SYSTEM temexdmodluyben
  (* Version 1.0, Author, 4DIAC-Consortium *)
  APPLICATION App1_ProdRateandPressure
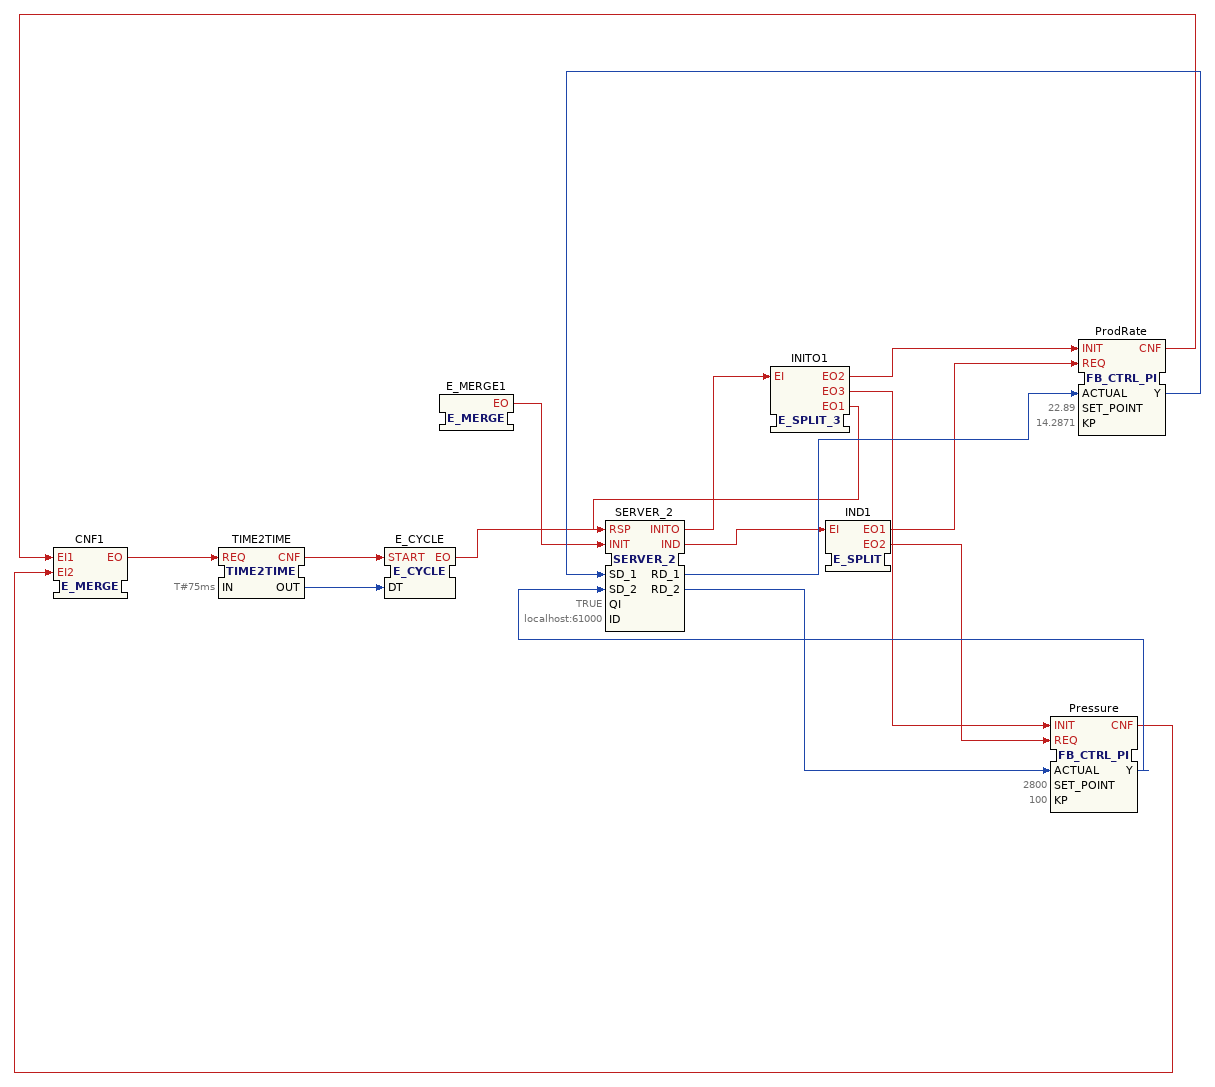
    FBS
      ProdRate : FB_CTRL_PI(SET_POINT := 22.89, KP := 14.2871);
      E_CYCLE : E_CYCLE;
      TIME2TIME : TIME2TIME(IN := T#75ms);
      SERVER_2 : SERVER_2(QI := TRUE, ID := localhost:61000);
      Pressure : FB_CTRL_PI(SET_POINT := 2800, KP := 100);
      INITO1 : E_SPLIT_3;
      IND1 : E_SPLIT;
      CNF1 : E_MERGE;
      E_MERGE1 : E_MERGE;
    END_FBS
    EVENT_CONNECTIONS
      TIME2TIME.CNF TO E_CYCLE.START;
      E_CYCLE.EO TO SERVER_2.RSP;
      SERVER_2.INITO TO INITO1.EI;
      INITO1.EO2 TO ProdRate.INIT;
      INITO1.EO3 TO Pressure.INIT;
      INITO1.EO1 TO SERVER_2.RSP;
      SERVER_2.IND TO IND1.EI;
      IND1.EO1 TO ProdRate.REQ;
      IND1.EO2 TO Pressure.REQ;
      ProdRate.CNF TO CNF1.EI1;
      Pressure.CNF TO CNF1.EI2;
      CNF1.EO TO TIME2TIME.REQ;
      E_MERGE1.EO TO SERVER_2.INIT;
    END_CONNECTIONS
    DATA_CONNECTIONS
      TIME2TIME.OUT TO E_CYCLE.DT;
      SERVER_2.RD_1 TO ProdRate.ACTUAL;
      SERVER_2.RD_2 TO Pressure.ACTUAL;
      ProdRate.Y TO SERVER_2.SD_1;
      Pressure.Y TO SERVER_2.SD_2;
    END_CONNECTIONS
  END_APPLICATION
  APPLICATION App2_StripperTemperatureandReactorTemperature
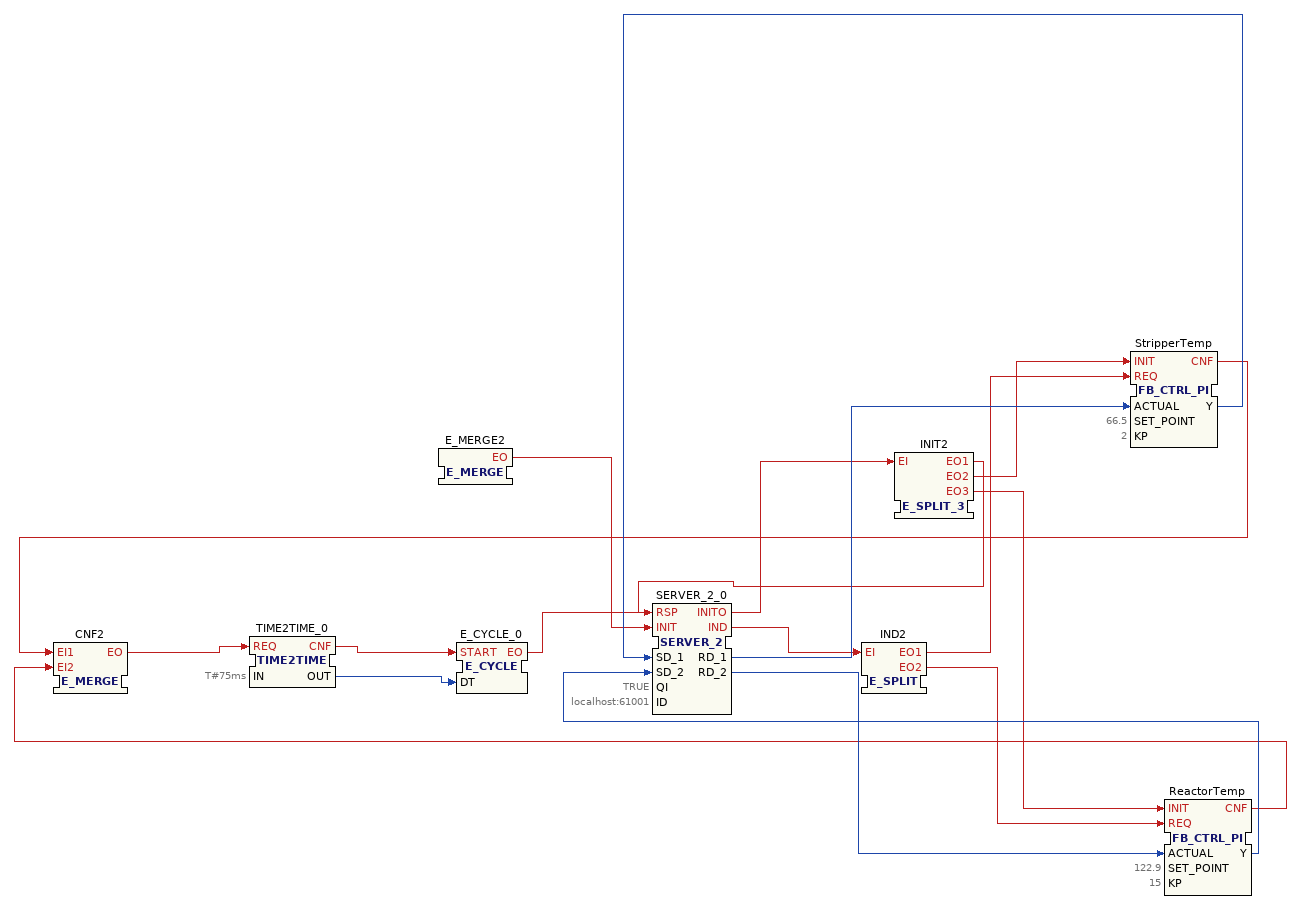
    FBS
      StripperTemp : FB_CTRL_PI(SET_POINT := 66.5, KP := 2);
      E_CYCLE_0 : E_CYCLE;
      TIME2TIME_0 : TIME2TIME(IN := T#75ms);
      SERVER_2_0 : SERVER_2(QI := TRUE, ID := localhost:61001);
      ReactorTemp : FB_CTRL_PI(SET_POINT := 122.9, KP := 15);
      CNF2 : E_MERGE;
      IND2 : E_SPLIT;
      INIT2 : E_SPLIT_3;
      E_MERGE2 : E_MERGE;
    END_FBS
    EVENT_CONNECTIONS
      E_CYCLE_0.EO TO SERVER_2_0.RSP;
      TIME2TIME_0.CNF TO E_CYCLE_0.START;
      SERVER_2_0.INITO TO INIT2.EI;
      INIT2.EO1 TO SERVER_2_0.RSP;
      INIT2.EO2 TO StripperTemp.INIT;
      INIT2.EO3 TO ReactorTemp.INIT;
      SERVER_2_0.IND TO IND2.EI;
      IND2.EO1 TO StripperTemp.REQ;
      IND2.EO2 TO ReactorTemp.REQ;
      StripperTemp.CNF TO CNF2.EI1;
      ReactorTemp.CNF TO CNF2.EI2;
      CNF2.EO TO TIME2TIME_0.REQ;
      E_MERGE2.EO TO SERVER_2_0.INIT;
    END_CONNECTIONS
    DATA_CONNECTIONS
      TIME2TIME_0.OUT TO E_CYCLE_0.DT;
      StripperTemp.Y TO SERVER_2_0.SD_1;
      SERVER_2_0.RD_1 TO StripperTemp.ACTUAL;
      SERVER_2_0.RD_2 TO ReactorTemp.ACTUAL;
      ReactorTemp.Y TO SERVER_2_0.SD_2;
    END_CONNECTIONS
  END_APPLICATION
  APPLICATION App3_StripperLevelandSeparatorLevel
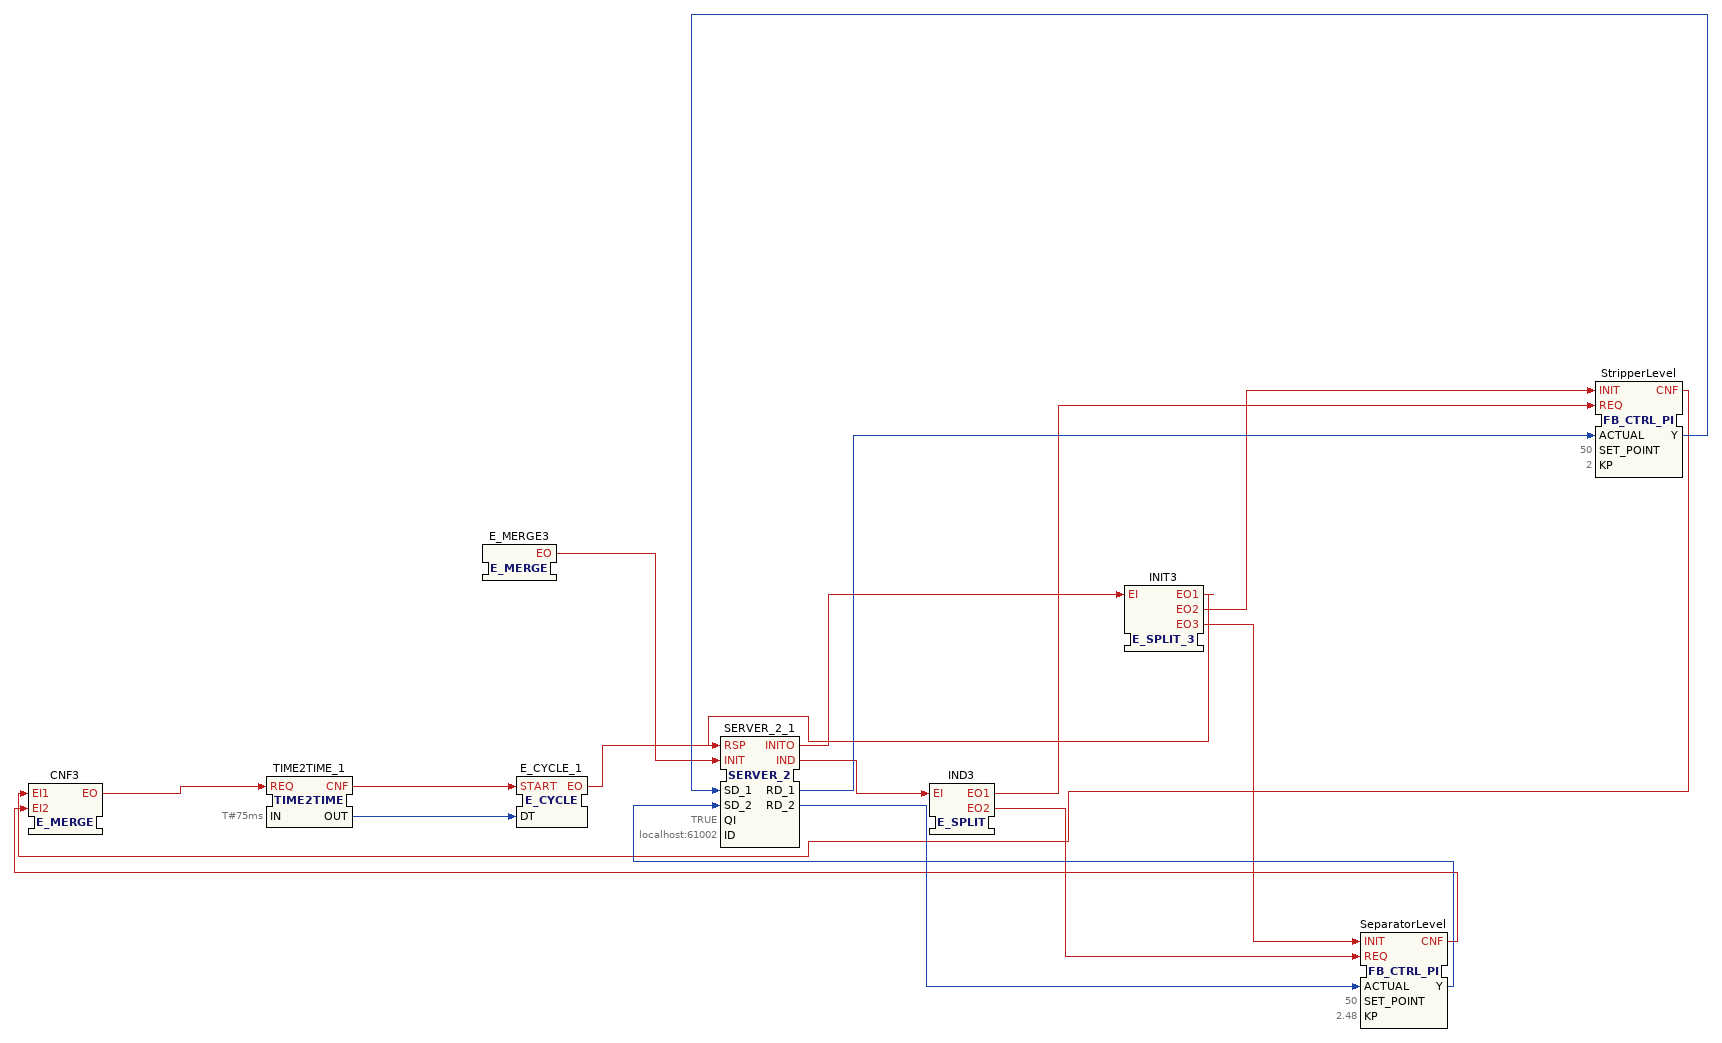
    FBS
      StripperLevel : FB_CTRL_PI(SET_POINT := 50, KP := 2);
      E_CYCLE_1 : E_CYCLE;
      TIME2TIME_1 : TIME2TIME(IN := T#75ms);
      SERVER_2_1 : SERVER_2(QI := TRUE, ID := localhost:61002);
      SeparatorLevel : FB_CTRL_PI(SET_POINT := 50, KP := 2.48);
      INIT3 : E_SPLIT_3;
      IND3 : E_SPLIT;
      CNF3 : E_MERGE;
      E_MERGE3 : E_MERGE;
    END_FBS
    EVENT_CONNECTIONS
      E_CYCLE_1.EO TO SERVER_2_1.RSP;
      TIME2TIME_1.CNF TO E_CYCLE_1.START;
      SERVER_2_1.INITO TO INIT3.EI;
      INIT3.EO1 TO SERVER_2_1.RSP;
      INIT3.EO2 TO StripperLevel.INIT;
      INIT3.EO3 TO SeparatorLevel.INIT;
      SERVER_2_1.IND TO IND3.EI;
      IND3.EO1 TO StripperLevel.REQ;
      IND3.EO2 TO SeparatorLevel.REQ;
      CNF3.EO TO TIME2TIME_1.REQ;
      StripperLevel.CNF TO CNF3.EI1;
      SeparatorLevel.CNF TO CNF3.EI2;
      E_MERGE3.EO TO SERVER_2_1.INIT;
    END_CONNECTIONS
    DATA_CONNECTIONS
      TIME2TIME_1.OUT TO E_CYCLE_1.DT;
      StripperLevel.Y TO SERVER_2_1.SD_1;
      SERVER_2_1.RD_1 TO StripperLevel.ACTUAL;
      SERVER_2_1.RD_2 TO SeparatorLevel.ACTUAL;
      SeparatorLevel.Y TO SERVER_2_1.SD_2;
    END_CONNECTIONS
  END_APPLICATION
  APPLICATION App4_ReactorLevel
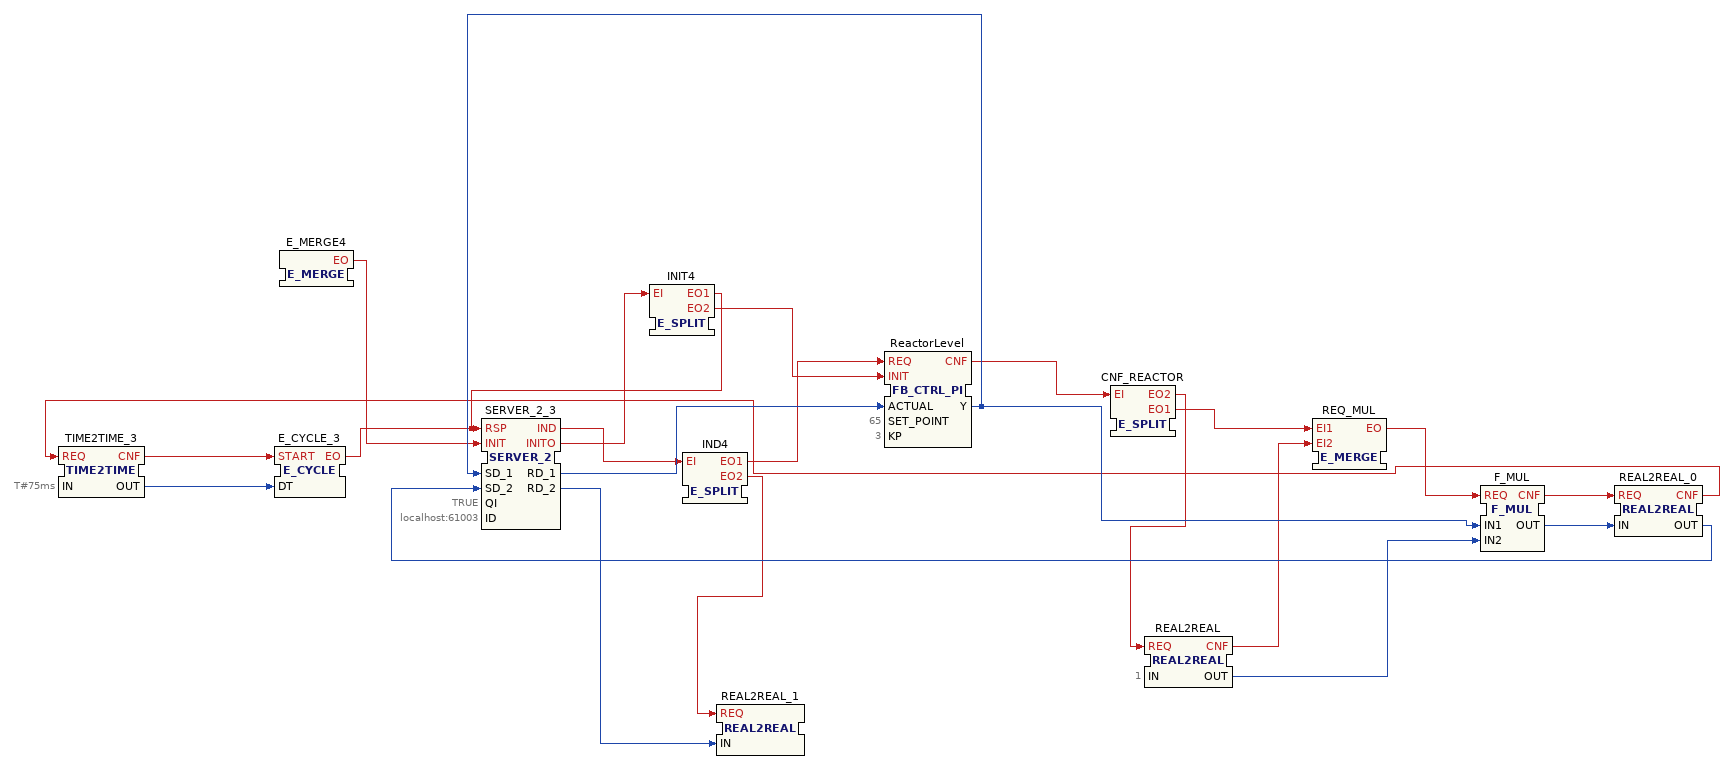
    FBS
      ReactorLevel : FB_CTRL_PI(SET_POINT := 65, KP := 3);
      E_CYCLE_3 : E_CYCLE;
      TIME2TIME_3 : TIME2TIME(IN := T#75ms);
      SERVER_2_3 : SERVER_2(QI := TRUE, ID := localhost:61003);
      F_MUL : F_MUL;
      REAL2REAL : REAL2REAL(IN := 1);
      REAL2REAL_0 : REAL2REAL;
      REAL2REAL_1 : REAL2REAL;
      IND4 : E_SPLIT;
      INIT4 : E_SPLIT;
      REQ_MUL : E_MERGE;
      CNF_REACTOR : E_SPLIT;
      E_MERGE4 : E_MERGE;
    END_FBS
    EVENT_CONNECTIONS
      E_CYCLE_3.EO TO SERVER_2_3.RSP;
      TIME2TIME_3.CNF TO E_CYCLE_3.START;
      F_MUL.CNF TO REAL2REAL_0.REQ;
      REAL2REAL_0.CNF TO TIME2TIME_3.REQ;
      SERVER_2_3.IND TO IND4.EI;
      IND4.EO1 TO ReactorLevel.REQ;
      IND4.EO2 TO REAL2REAL_1.REQ;
      SERVER_2_3.INITO TO INIT4.EI;
      INIT4.EO1 TO SERVER_2_3.RSP;
      INIT4.EO2 TO ReactorLevel.INIT;
      ReactorLevel.CNF TO CNF_REACTOR.EI;
      CNF_REACTOR.EO2 TO REAL2REAL.REQ;
      CNF_REACTOR.EO1 TO REQ_MUL.EI1;
      REAL2REAL.CNF TO REQ_MUL.EI2;
      REQ_MUL.EO TO F_MUL.REQ;
      E_MERGE4.EO TO SERVER_2_3.INIT;
    END_CONNECTIONS
    DATA_CONNECTIONS
      TIME2TIME_3.OUT TO E_CYCLE_3.DT;
      ReactorLevel.Y TO SERVER_2_3.SD_1;
      SERVER_2_3.RD_1 TO ReactorLevel.ACTUAL;
      ReactorLevel.Y TO F_MUL.IN1;
      REAL2REAL.OUT TO F_MUL.IN2;
      F_MUL.OUT TO REAL2REAL_0.IN;
      REAL2REAL_0.OUT TO SERVER_2_3.SD_2;
      SERVER_2_3.RD_2 TO REAL2REAL_1.IN;
    END_CONNECTIONS
  END_APPLICATION
  APPLICATION App5_yAandyB
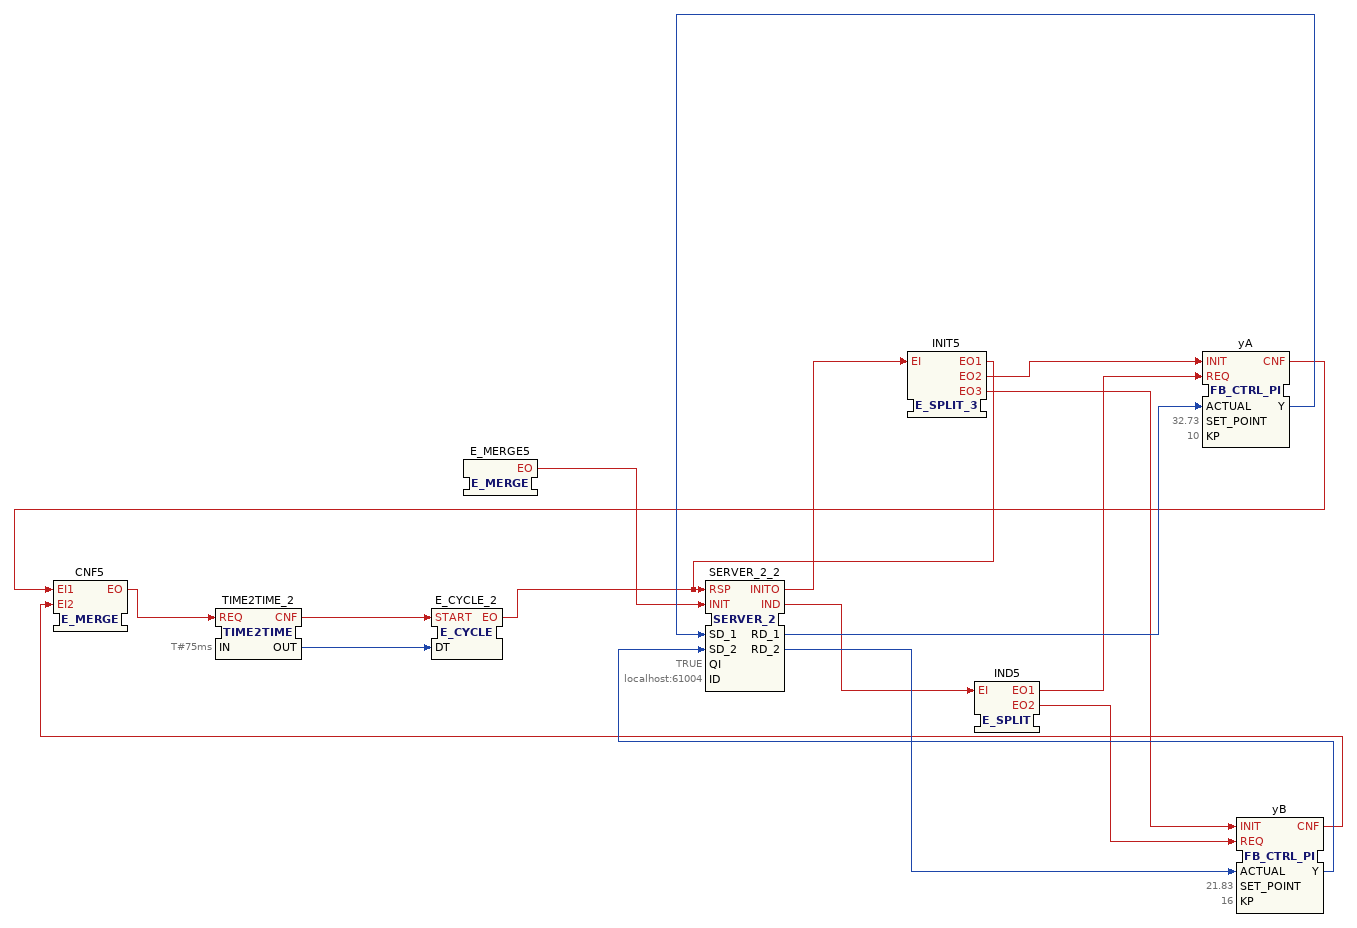
    FBS
      yA : FB_CTRL_PI(SET_POINT := 32.73, KP := 10);
      E_CYCLE_2 : E_CYCLE;
      TIME2TIME_2 : TIME2TIME(IN := T#75ms);
      SERVER_2_2 : SERVER_2(QI := TRUE, ID := localhost:61004);
      yB : FB_CTRL_PI(SET_POINT := 21.83, KP := 16);
      INIT5 : E_SPLIT_3;
      IND5 : E_SPLIT;
      CNF5 : E_MERGE;
      E_MERGE5 : E_MERGE;
    END_FBS
    EVENT_CONNECTIONS
      E_CYCLE_2.EO TO SERVER_2_2.RSP;
      TIME2TIME_2.CNF TO E_CYCLE_2.START;
      SERVER_2_2.INITO TO INIT5.EI;
      INIT5.EO1 TO SERVER_2_2.RSP;
      INIT5.EO2 TO yA.INIT;
      INIT5.EO3 TO yB.INIT;
      SERVER_2_2.IND TO IND5.EI;
      IND5.EO1 TO yA.REQ;
      IND5.EO2 TO yB.REQ;
      CNF5.EO TO TIME2TIME_2.REQ;
      yA.CNF TO CNF5.EI1;
      yB.CNF TO CNF5.EI2;
      E_MERGE5.EO TO SERVER_2_2.INIT;
    END_CONNECTIONS
    DATA_CONNECTIONS
      TIME2TIME_2.OUT TO E_CYCLE_2.DT;
      yA.Y TO SERVER_2_2.SD_1;
      SERVER_2_2.RD_1 TO yA.ACTUAL;
      SERVER_2_2.RD_2 TO yB.ACTUAL;
      yB.Y TO SERVER_2_2.SD_2;
    END_CONNECTIONS
  END_APPLICATION
  DEVICE FORTE_PC : FORTE_PC(MGR_ID := "localhost:61499")
    {SET_ATTRIBUTE(Profile, HOLOBLOC)}
    RESOURCE EMB_RES : EMB_RES
      FBS
        ProdRate : FB_CTRL_PI(SET_POINT := 22.89, KP := 14.2871);
        E_CYCLE : E_CYCLE;
        TIME2TIME : TIME2TIME(IN := T#75ms);
        SERVER_2 : SERVER_2(QI := TRUE, ID := localhost:61000);
        Pressure : FB_CTRL_PI(SET_POINT := 2800, KP := 100);
        StripperTemp : FB_CTRL_PI(SET_POINT := 66.5, KP := 2);
        E_CYCLE_0 : E_CYCLE;
        TIME2TIME_0 : TIME2TIME(IN := T#75ms);
        SERVER_2_0 : SERVER_2(QI := TRUE, ID := localhost:61001);
        ReactorTemp : FB_CTRL_PI(SET_POINT := 122.9, KP := 15);
        ReactorLevel : FB_CTRL_PI(SET_POINT := 65, KP := 3);
        E_CYCLE_3 : E_CYCLE;
        TIME2TIME_3 : TIME2TIME(IN := T#75ms);
        SERVER_2_3 : SERVER_2(QI := TRUE, ID := localhost:61003);
        F_MUL : F_MUL;
        REAL2REAL : REAL2REAL(IN := 1);
        REAL2REAL_0 : REAL2REAL;
        REAL2REAL_1 : REAL2REAL;
        yA : FB_CTRL_PI(SET_POINT := 32.73, KP := 10);
        E_CYCLE_2 : E_CYCLE;
        TIME2TIME_2 : TIME2TIME(IN := T#75ms);
        SERVER_2_2 : SERVER_2(QI := TRUE, ID := localhost:61004);
        yB : FB_CTRL_PI(SET_POINT := 21.83, KP := 16);
        StripperLevel : FB_CTRL_PI(SET_POINT := 50, KP := 2);
        E_CYCLE_1 : E_CYCLE;
        TIME2TIME_1 : TIME2TIME(IN := T#75ms);
        SERVER_2_1 : SERVER_2(QI := TRUE, ID := localhost:61002);
        SeparatorLevel : FB_CTRL_PI(SET_POINT := 50, KP := 2.48);
        CNF1 : E_MERGE;
        IND1 : E_SPLIT;
        INITO1 : E_SPLIT_3;
        CNF2 : E_MERGE;
        INIT2 : E_SPLIT_3;
        IND2 : E_SPLIT;
        IND3 : E_SPLIT;
        INIT3 : E_SPLIT_3;
        CNF3 : E_MERGE;
        IND4 : E_SPLIT;
        INIT4 : E_SPLIT;
        CNF_REACTOR : E_SPLIT;
        REQ_MUL : E_MERGE;
        INIT5 : E_SPLIT_3;
        IND5 : E_SPLIT;
        CNF5 : E_MERGE;
        E_SPLIT_5 : E_SPLIT_5;
        E_SPLIT_5_0 : E_SPLIT_5;
        E_MERGE1 : E_MERGE;
        E_MERGE2 : E_MERGE;
        E_MERGE3 : E_MERGE;
        E_MERGE5 : E_MERGE;
        E_MERGE4 : E_MERGE;
      END_FBS
      EVENT_CONNECTIONS
        TIME2TIME.CNF TO E_CYCLE.START;
        E_CYCLE.EO TO SERVER_2.RSP;
        TIME2TIME_0.CNF TO E_CYCLE_0.START;
        E_CYCLE_0.EO TO SERVER_2_0.RSP;
        TIME2TIME_3.CNF TO E_CYCLE_3.START;
        E_CYCLE_3.EO TO SERVER_2_3.RSP;
        F_MUL.CNF TO REAL2REAL_0.REQ;
        REAL2REAL_0.CNF TO TIME2TIME_3.REQ;
        TIME2TIME_2.CNF TO E_CYCLE_2.START;
        E_CYCLE_2.EO TO SERVER_2_2.RSP;
        TIME2TIME_1.CNF TO E_CYCLE_1.START;
        E_CYCLE_1.EO TO SERVER_2_1.RSP;
        ProdRate.CNF TO CNF1.EI1;
        Pressure.CNF TO CNF1.EI2;
        CNF1.EO TO TIME2TIME.REQ;
        SERVER_2.IND TO IND1.EI;
        IND1.EO1 TO ProdRate.REQ;
        IND1.EO2 TO Pressure.REQ;
        SERVER_2.INITO TO INITO1.EI;
        INITO1.EO1 TO SERVER_2.RSP;
        INITO1.EO2 TO ProdRate.INIT;
        INITO1.EO3 TO Pressure.INIT;
        StripperTemp.CNF TO CNF2.EI1;
        ReactorTemp.CNF TO CNF2.EI2;
        CNF2.EO TO TIME2TIME_0.REQ;
        SERVER_2_0.INITO TO INIT2.EI;
        INIT2.EO1 TO SERVER_2_0.RSP;
        INIT2.EO2 TO StripperTemp.INIT;
        INIT2.EO3 TO ReactorTemp.INIT;
        SERVER_2_0.IND TO IND2.EI;
        IND2.EO1 TO StripperTemp.REQ;
        IND2.EO2 TO ReactorTemp.REQ;
        SERVER_2_1.IND TO IND3.EI;
        IND3.EO1 TO StripperLevel.REQ;
        IND3.EO2 TO SeparatorLevel.REQ;
        SERVER_2_1.INITO TO INIT3.EI;
        INIT3.EO1 TO SERVER_2_1.RSP;
        INIT3.EO2 TO StripperLevel.INIT;
        INIT3.EO3 TO SeparatorLevel.INIT;
        StripperLevel.CNF TO CNF3.EI1;
        SeparatorLevel.CNF TO CNF3.EI2;
        CNF3.EO TO TIME2TIME_1.REQ;
        SERVER_2_3.IND TO IND4.EI;
        IND4.EO1 TO ReactorLevel.REQ;
        IND4.EO2 TO REAL2REAL_1.REQ;
        SERVER_2_3.INITO TO INIT4.EI;
        INIT4.EO1 TO SERVER_2_3.RSP;
        INIT4.EO2 TO ReactorLevel.INIT;
        ReactorLevel.CNF TO CNF_REACTOR.EI;
        CNF_REACTOR.EO2 TO REAL2REAL.REQ;
        CNF_REACTOR.EO1 TO REQ_MUL.EI1;
        REAL2REAL.CNF TO REQ_MUL.EI2;
        REQ_MUL.EO TO F_MUL.REQ;
        SERVER_2_2.INITO TO INIT5.EI;
        INIT5.EO1 TO SERVER_2_2.RSP;
        INIT5.EO2 TO yA.INIT;
        INIT5.EO3 TO yB.INIT;
        SERVER_2_2.IND TO IND5.EI;
        IND5.EO1 TO yA.REQ;
        IND5.EO2 TO yB.REQ;
        yA.CNF TO CNF5.EI1;
        yB.CNF TO CNF5.EI2;
        CNF5.EO TO TIME2TIME_2.REQ;
        START.COLD TO E_SPLIT_5.EI;
        START.WARM TO E_SPLIT_5_0.EI;
        E_MERGE1.EO TO SERVER_2.INIT;
        E_MERGE2.EO TO SERVER_2_0.INIT;
        E_MERGE3.EO TO SERVER_2_1.INIT;
        E_MERGE5.EO TO SERVER_2_2.INIT;
        E_MERGE4.EO TO SERVER_2_3.INIT;
        E_SPLIT_5.EO1 TO E_MERGE1.EI1;
        E_SPLIT_5_0.EO1 TO E_MERGE1.EI2;
        E_SPLIT_5.EO2 TO E_MERGE2.EI1;
        E_SPLIT_5_0.EO2 TO E_MERGE2.EI2;
        E_SPLIT_5.EO3 TO E_MERGE3.EI1;
        E_SPLIT_5_0.EO3 TO E_MERGE3.EI2;
        E_SPLIT_5.EO4 TO E_MERGE4.EI1;
        E_SPLIT_5_0.EO4 TO E_MERGE4.EI2;
        E_SPLIT_5.EO5 TO E_MERGE5.EI1;
        E_SPLIT_5_0.EO5 TO E_MERGE5.EI2;
      END_CONNECTIONS
      DATA_CONNECTIONS
        TIME2TIME.OUT TO E_CYCLE.DT;
        ProdRate.Y TO SERVER_2.SD_1;
        SERVER_2.RD_1 TO ProdRate.ACTUAL;
        SERVER_2.RD_2 TO Pressure.ACTUAL;
        Pressure.Y TO SERVER_2.SD_2;
        TIME2TIME_0.OUT TO E_CYCLE_0.DT;
        StripperTemp.Y TO SERVER_2_0.SD_1;
        SERVER_2_0.RD_1 TO StripperTemp.ACTUAL;
        SERVER_2_0.RD_2 TO ReactorTemp.ACTUAL;
        ReactorTemp.Y TO SERVER_2_0.SD_2;
        TIME2TIME_3.OUT TO E_CYCLE_3.DT;
        ReactorLevel.Y TO SERVER_2_3.SD_1;
        SERVER_2_3.RD_1 TO ReactorLevel.ACTUAL;
        ReactorLevel.Y TO F_MUL.IN1;
        REAL2REAL.OUT TO F_MUL.IN2;
        F_MUL.OUT TO REAL2REAL_0.IN;
        REAL2REAL_0.OUT TO SERVER_2_3.SD_2;
        SERVER_2_3.RD_2 TO REAL2REAL_1.IN;
        TIME2TIME_2.OUT TO E_CYCLE_2.DT;
        yA.Y TO SERVER_2_2.SD_1;
        SERVER_2_2.RD_1 TO yA.ACTUAL;
        SERVER_2_2.RD_2 TO yB.ACTUAL;
        yB.Y TO SERVER_2_2.SD_2;
        TIME2TIME_1.OUT TO E_CYCLE_1.DT;
        StripperLevel.Y TO SERVER_2_1.SD_1;
        SERVER_2_1.RD_1 TO StripperLevel.ACTUAL;
        SERVER_2_1.RD_2 TO SeparatorLevel.ACTUAL;
        SeparatorLevel.Y TO SERVER_2_1.SD_2;
      END_CONNECTIONS
    END_RESOURCE
  END_DEVICE
  MAPPINGS
    App1_ProdRateandPressure.ProdRate ON FORTE_PC.EMB_RES.ProdRate;
    App1_ProdRateandPressure.E_CYCLE ON FORTE_PC.EMB_RES.E_CYCLE;
    App1_ProdRateandPressure.TIME2TIME ON FORTE_PC.EMB_RES.TIME2TIME;
    App1_ProdRateandPressure.SERVER_2 ON FORTE_PC.EMB_RES.SERVER_2;
    App1_ProdRateandPressure.Pressure ON FORTE_PC.EMB_RES.Pressure;
    App1_ProdRateandPressure.INITO1 ON FORTE_PC.EMB_RES.INITO1;
    App1_ProdRateandPressure.IND1 ON FORTE_PC.EMB_RES.IND1;
    App1_ProdRateandPressure.CNF1 ON FORTE_PC.EMB_RES.CNF1;
    App1_ProdRateandPressure.E_MERGE1 ON FORTE_PC.EMB_RES.E_MERGE1;
    App2_StripperTemperatureandReactorTemperature.StripperTemp ON FORTE_PC.EMB_RES.StripperTemp;
    App2_StripperTemperatureandReactorTemperature.E_CYCLE_0 ON FORTE_PC.EMB_RES.E_CYCLE_0;
    App2_StripperTemperatureandReactorTemperature.TIME2TIME_0 ON FORTE_PC.EMB_RES.TIME2TIME_0;
    App2_StripperTemperatureandReactorTemperature.SERVER_2_0 ON FORTE_PC.EMB_RES.SERVER_2_0;
    App2_StripperTemperatureandReactorTemperature.ReactorTemp ON FORTE_PC.EMB_RES.ReactorTemp;
    App2_StripperTemperatureandReactorTemperature.CNF2 ON FORTE_PC.EMB_RES.CNF2;
    App2_StripperTemperatureandReactorTemperature.IND2 ON FORTE_PC.EMB_RES.IND2;
    App2_StripperTemperatureandReactorTemperature.INIT2 ON FORTE_PC.EMB_RES.INIT2;
    App2_StripperTemperatureandReactorTemperature.E_MERGE2 ON FORTE_PC.EMB_RES.E_MERGE2;
    App3_StripperLevelandSeparatorLevel.StripperLevel ON FORTE_PC.EMB_RES.StripperLevel;
    App3_StripperLevelandSeparatorLevel.E_CYCLE_1 ON FORTE_PC.EMB_RES.E_CYCLE_1;
    App3_StripperLevelandSeparatorLevel.TIME2TIME_1 ON FORTE_PC.EMB_RES.TIME2TIME_1;
    App3_StripperLevelandSeparatorLevel.SERVER_2_1 ON FORTE_PC.EMB_RES.SERVER_2_1;
    App3_StripperLevelandSeparatorLevel.SeparatorLevel ON FORTE_PC.EMB_RES.SeparatorLevel;
    App3_StripperLevelandSeparatorLevel.INIT3 ON FORTE_PC.EMB_RES.INIT3;
    App3_StripperLevelandSeparatorLevel.IND3 ON FORTE_PC.EMB_RES.IND3;
    App3_StripperLevelandSeparatorLevel.CNF3 ON FORTE_PC.EMB_RES.CNF3;
    App3_StripperLevelandSeparatorLevel.E_MERGE3 ON FORTE_PC.EMB_RES.E_MERGE3;
    App4_ReactorLevel.ReactorLevel ON FORTE_PC.EMB_RES.ReactorLevel;
    App4_ReactorLevel.E_CYCLE_3 ON FORTE_PC.EMB_RES.E_CYCLE_3;
    App4_ReactorLevel.TIME2TIME_3 ON FORTE_PC.EMB_RES.TIME2TIME_3;
    App4_ReactorLevel.SERVER_2_3 ON FORTE_PC.EMB_RES.SERVER_2_3;
    App4_ReactorLevel.F_MUL ON FORTE_PC.EMB_RES.F_MUL;
    App4_ReactorLevel.REAL2REAL ON FORTE_PC.EMB_RES.REAL2REAL;
    App4_ReactorLevel.REAL2REAL_0 ON FORTE_PC.EMB_RES.REAL2REAL_0;
    App4_ReactorLevel.REAL2REAL_1 ON FORTE_PC.EMB_RES.REAL2REAL_1;
    App4_ReactorLevel.IND4 ON FORTE_PC.EMB_RES.IND4;
    App4_ReactorLevel.INIT4 ON FORTE_PC.EMB_RES.INIT4;
    App4_ReactorLevel.REQ_MUL ON FORTE_PC.EMB_RES.REQ_MUL;
    App4_ReactorLevel.CNF_REACTOR ON FORTE_PC.EMB_RES.CNF_REACTOR;
    App4_ReactorLevel.E_MERGE4 ON FORTE_PC.EMB_RES.E_MERGE4;
    App5_yAandyB.yA ON FORTE_PC.EMB_RES.yA;
    App5_yAandyB.E_CYCLE_2 ON FORTE_PC.EMB_RES.E_CYCLE_2;
    App5_yAandyB.TIME2TIME_2 ON FORTE_PC.EMB_RES.TIME2TIME_2;
    App5_yAandyB.SERVER_2_2 ON FORTE_PC.EMB_RES.SERVER_2_2;
    App5_yAandyB.yB ON FORTE_PC.EMB_RES.yB;
    App5_yAandyB.INIT5 ON FORTE_PC.EMB_RES.INIT5;
    App5_yAandyB.IND5 ON FORTE_PC.EMB_RES.IND5;
    App5_yAandyB.CNF5 ON FORTE_PC.EMB_RES.CNF5;
    App5_yAandyB.E_MERGE5 ON FORTE_PC.EMB_RES.E_MERGE5;
  END_MAPPINGS
  SEGMENTS
    Ethernet : Ethernet;
  END_SEGMENTS
  LINKS
    FORTE_PC => Ethernet;
  END_LINKS
END_SYSTEM
